FUNCTION_BLOCK FB_SolenoidControl
VAR_INPUT
    bExecute      : BOOL;  			// Activates control of solenoid valves
    eSolenoidSet  : E_SolenoidSet; 	// Enum with valve configuration
END_VAR

VAR_OUTPUT
    bDone         : BOOL;  			// Indicates that the valves have been positioned correctly
END_VAR

VAR
    eState        : (IDLE, SET_VALVES, DONE);
END_VAR

CASE eState OF
    IDLE:
        IF bExecute THEN
            eState := SET_VALVES;
        END_IF;

    SET_VALVES: //Setting position accordantly pneumatics drawnings for Solenoid Valves A, B e C. 
        CASE eSolenoidSet OF
            E_SolenoidSet.IDLE:
                GVL_IO.gDigOutputs.bSolenoidValveA := FALSE;
                GVL_IO.gDigOutputs.bSolenoidValveB := FALSE;
                GVL_IO.gDigOutputs.bSolenoidValveC := FALSE;
            E_SolenoidSet.LEAKTEST:
                GVL_IO.gDigOutputs.bSolenoidValveA := FALSE;
                GVL_IO.gDigOutputs.bSolenoidValveB := TRUE;
                GVL_IO.gDigOutputs.bSolenoidValveC := FALSE;
           E_SolenoidSet.LEAKTESTMONITORING:
                GVL_IO.gDigOutputs.bSolenoidValveA := TRUE;
                GVL_IO.gDigOutputs.bSolenoidValveB := FALSE;
                GVL_IO.gDigOutputs.bSolenoidValveC := FALSE;
            E_SolenoidSet.AIRDRY:
                GVL_IO.gDigOutputs.bSolenoidValveA := FALSE;
                GVL_IO.gDigOutputs.bSolenoidValveB := FALSE;
                GVL_IO.gDigOutputs.bSolenoidValveC := TRUE;
        END_CASE;
        eState := DONE;
    
    DONE:
        bDone := TRUE;
END_CASE;

END_FUNCTION_BLOCK

(* stored: Version 1.1.0.1, ProductVersion 3.1.4024.12
   POU FB_SolenoidControl: Id {6fdcc804-c623-4349-8517-cdc349f41989}, SpecialFunc None *)
